INTERFACE I_terminal_execution

METHOD run : BOOL
VAR_INPUT
END_VAR
END_METHOD

END_INTERFACE

(* stored: Version 1.1.0.1, ProductVersion 3.1.4024.6
   Itf I_terminal_execution: Id {1013d006-3a3b-0bdf-1cfb-2a9b89f221d5}
   Method run: Id {cff3d69d-5408-0591-120d-452081181024} *)
